FUNCTION_BLOCK FB_TheThing
VAR_INPUT
	input	: REAL;
END_VAR
VAR_OUTPUT
	output	: REAL;
END_VAR
VAR

	prepared			: BOOL := FALSE;
	succeeded			: BOOL := FALSE;
	
	preparation_timer	: TON;
	
	offset				: REAL := 0;
	testAdd				: BOOL;
	
END_VAR


prepared := prepare_to_do_the_thing();

succeeded := do_the_thing();

METHOD do_the_thing : BOOL
VAR_INPUT
END_VAR
THIS^.output := SEL(THIS^.prepared, 0, input - THIS^.offset);

do_the_thing := NOT THIS^.prepared;
END_METHOD

METHOD prepare_to_do_the_thing : BOOL
VAR_INPUT

END_VAR
preparation_timer(IN := NOT THIS^.prepared, PT := T#3S);

THIS^.offset := SEL(preparation_timer.Q, THIS^.offset, (THIS^.offset + input) / 2);

prepare_to_do_the_thing := preparation_timer.Q;
END_METHOD

END_FUNCTION_BLOCK

(* stored: Version 1.1.0.1, ProductVersion 3.1.4022.18
   POU FB_TheThing: Id {ae585d05-c753-4c3e-90dd-c6220bf5bb9e}, SpecialFunc None
   Method do_the_thing: Id {407deb4a-f778-4693-9eec-d23695a1fdb0}
   Method prepare_to_do_the_thing: Id {c175b9c6-84df-458d-abed-deba4a8f659f} *)
